{attribute 'qualified_only'}
VAR_GLOBAL
	rand_generator: DRAND := (Seed := 154);
END_VAR

(* stored: Version 1.1.0.1, ProductVersion 3.1.4026.0
   GVL GVL: Id {40b54f84-49ac-499b-abab-103d39a49576} *)
